SUBAPPLICATION Uebung_021_AX (* Spiegelabfolge (1) - AX Variante *)
  (* Standard: 61499-2; Description: Copyright (c) 2023 Meisterschulen am Ostbahnhof This program and the accompanying materials are made available under the terms of the Eclipse Public License 2.0 which is available at https://www.eclipse.org/legal/epl-2.0/ SPDX-License-Identifier: EPL-2.0 *)
  (* Version 1.0, 2026-04-20, Franz Höpfinger, Meisterschulen am Ostbahnhof, AX Variante *)
  PACKAGE Uebungen;
  IMPORT Uebungen::const::UT::DefaultPool::SoftKey_F1;
  IMPORT Uebungen::const::UT::DefaultPool::SoftKey_F2;
  IMPORT logiBUS::io::DQ::logiBUS_DO::Output_Q1;
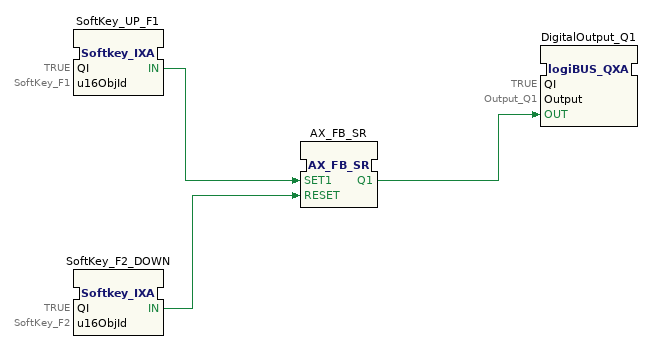
  (* START-Knopf *)
  (* Endlage *)
  FBS
    DigitalOutput_Q1 : logiBUS::io::DQ::logiBUS_QXA(QI := TRUE, Output := Output_Q1);
    SoftKey_UP_F1 : isobus::UT::io::Softkey::Softkey_IXA(QI := TRUE, u16ObjId := SoftKey_F1);
    AX_FB_SR : adapter::iec61131::bistableElements::AX_FB_SR;
    SoftKey_F2_DOWN : isobus::UT::io::Softkey::Softkey_IXA(QI := TRUE, u16ObjId := SoftKey_F2);
  END_FBS
  ADAPTER_CONNECTIONS
    AX_FB_SR.Q1 TO DigitalOutput_Q1.OUT;
    SoftKey_UP_F1.IN TO AX_FB_SR.SET1;
    SoftKey_F2_DOWN.IN TO AX_FB_SR.RESET;
  END_CONNECTIONS
END_SUBAPPLICATION
